// TIA Portal V17 export
// export: Created 2025-03-05T07:59:04.2255754Z, ExportSetting WithDefaults, DisplayName Totally Integrated Automation Portal, DisplayVersion V17 Update 8, DisplayName TIA Portal Openness, DisplayVersion V17 Update 8, DisplayName TIA Portal Version Control Interface, DisplayVersion V17, DisplayName SINAMICS Startdrive Advanced, DisplayVersion V17 SP2, DisplayName SINAMICS Startdrive G110M, G120, G120C, G120D, G120P, G115D, DisplayVersion V17 SP2, DisplayName SINAMICS Startdrive G130, G150, S120, S150, SINAMICS MV, S210, DisplayVersion V17 SP2, DisplayName STEP 7 Professional, DisplayVersion V17 Update 8, DisplayName SINUMERIK ONE STEP 7 Toolbox, DisplayVersion V17 Update 12, DisplayName SINUMERIK 840D sl STEP 7 Toolbox, DisplayVersion V17 Update 12, DisplayName STEP 7 Safety, DisplayVersion V17 Update 6, DisplayName WinCC Advanced, DisplayVersion V17 Update 8
FUNCTION_BLOCK "FB2502_PART_DETECTION_SENSOR"   // FB2502, LAD
{ S7_Optimized_Access := 'FALSE' }
AUTHOR : ETXETAR
VERSION : 1.0
// stored: AutoNumber false, IsIECCheckEnabled false, SetENOAutomatically false, UDAEnableTagReadback false
   VAR_INPUT
      INPUT : Word;   // INPUT
   END_VAR
   VAR_OUTPUT
      PART_PRESENT_FACE_A : Bool;   // CLAMPED WITHOUT PARTS / PART PRESENT FACE A UP
      PART_PRESENT_FACE_B : Bool;   // CLAMPED WITH PART / PART PRESENT FACE B UP
      PART_PRESENT : Bool;   // CLAMPED / PART_PRESENT
      NO_PART_PRESENT : Bool;   // UNCLAMPED / NO PART PRESENT
   END_VAR
   VAR DB_SPECIFIC
      CURRENT_VALUE { S7_SetPoint := 'True'} : DInt;   // CURRENT VALUE
      PART_FACE_A_PRESENT_MAX { S7_SetPoint := 'True'} : DInt;   // CLAMP MAX WITHOUT
      PART_FACE_A_PRESENT_MIN { S7_SetPoint := 'True'} : DInt := DINT#-10000;   // CLAMP MIN WITHOUT
      PART_FACE_B_PRESENT_MAX { S7_SetPoint := 'True'} : DInt := DINT#-10000;   // CLAMP MAX WITH
      PART_FACE_B_PRESENT_MIN { S7_SetPoint := 'True'} : DInt := DINT#-10000;   // CLAMP MIN WITH
      NO_PART_PRESENT_MAX { S7_SetPoint := 'True'} : DInt := DINT#-10000;   // UNCLAMP MAX
      NO_PART_PRESENT_MIN { S7_SetPoint := 'True'} : DInt := DINT#-10000;   // UNCLAMP MIN
   END_VAR
BEGIN

REGION Network 1: INPUTS
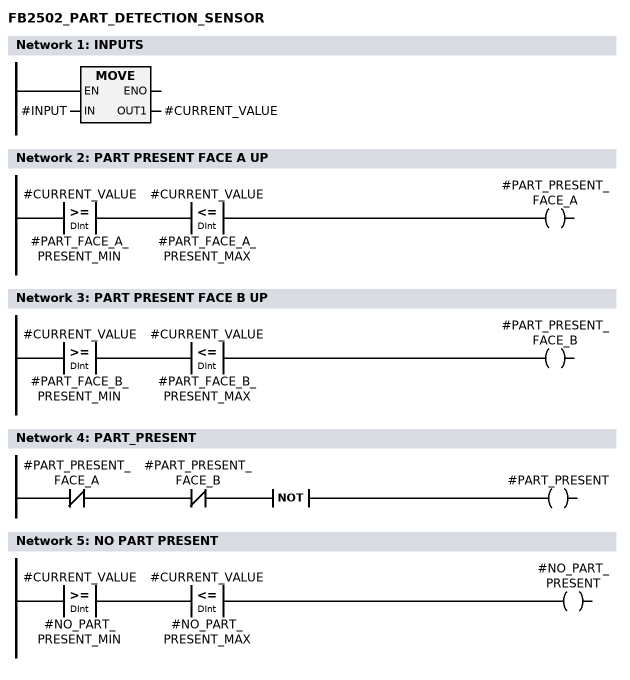
   RUNG wire#powerrail
      { S7_GenerateENO := "TRUE" } Move(in := #INPUT, out1 => #CURRENT_VALUE)
   END_RUNG
   // the same network as SCL:
   #CURRENT_VALUE := #INPUT;
END_REGION

REGION Network 2: PART PRESENT FACE A UP
   RUNG wire#powerrail
      { S7_Templates := "SrcType := DInt" } GE_Contact(in1 := #CURRENT_VALUE, in2 := #PART_FACE_A_PRESENT_MIN)
      { S7_Templates := "SrcType := DInt" } LE_Contact(in1 := #CURRENT_VALUE, in2 := #PART_FACE_A_PRESENT_MAX)
      Coil( #PART_PRESENT_FACE_A )
   END_RUNG
   // the same network as SCL:
   #PART_PRESENT_FACE_A := (#CURRENT_VALUE >= #PART_FACE_A_PRESENT_MIN) AND (#CURRENT_VALUE <= #PART_FACE_A_PRESENT_MAX);
END_REGION

REGION Network 3: PART PRESENT FACE B UP
   RUNG wire#powerrail
      { S7_Templates := "SrcType := DInt" } GE_Contact(in1 := #CURRENT_VALUE, in2 := #PART_FACE_B_PRESENT_MIN)
      { S7_Templates := "SrcType := DInt" } LE_Contact(in1 := #CURRENT_VALUE, in2 := #PART_FACE_B_PRESENT_MAX)
      Coil( #PART_PRESENT_FACE_B )
   END_RUNG
   // the same network as SCL:
   #PART_PRESENT_FACE_B := (#CURRENT_VALUE >= #PART_FACE_B_PRESENT_MIN) AND (#CURRENT_VALUE <= #PART_FACE_B_PRESENT_MAX);
END_REGION

REGION Network 4: PART_PRESENT
   RUNG wire#powerrail
      I_Contact( #PART_PRESENT_FACE_A )
      I_Contact( #PART_PRESENT_FACE_B )
      Not()
      Coil( #PART_PRESENT )
   END_RUNG
   // the same network as SCL:
   #PART_PRESENT := NOT (NOT #PART_PRESENT_FACE_A AND NOT #PART_PRESENT_FACE_B);
END_REGION

REGION Network 5: NO PART PRESENT
   RUNG wire#powerrail
      { S7_Templates := "SrcType := DInt" } GE_Contact(in1 := #CURRENT_VALUE, in2 := #NO_PART_PRESENT_MIN)
      { S7_Templates := "SrcType := DInt" } LE_Contact(in1 := #CURRENT_VALUE, in2 := #NO_PART_PRESENT_MAX)
      Coil( #NO_PART_PRESENT )
   END_RUNG
   // the same network as SCL:
   #NO_PART_PRESENT := (#CURRENT_VALUE >= #NO_PART_PRESENT_MIN) AND (#CURRENT_VALUE <= #NO_PART_PRESENT_MAX);
END_REGION
END_FUNCTION_BLOCK
